TYPE ST_ReadAllOffsetDataCommand EXTENDS ST_CommandBasic:
STRUCT
END_STRUCT
END_TYPE

(* stored: Version 1.1.0.1, ProductVersion 3.1.4024.13
   DUT ST_ReadAllOffsetDataCommand: Id {4bebd1ca-a693-4e9a-b4fa-f7d72c5e7809} *)
